# EPICS autosave request: ioc/autoSaveRestore/rampSetting.req
$(P)RampStepSize
$(P)RampInterval
$(P)TargetHV
$(P)RampMode
$(P)RampDuration
$(P)DeviceNickname
